(* IEC 61131-3 sources: exOS-Demos/Frameworks/Components/Binary/Sequence/Sequence, 2 files *)

(* ---- Sequence.typ ---- *)
TYPE
	SequenceButtons : 	STRUCT
		ButtonLeft : BOOL;
		ButtonRight : BOOL;
	END_STRUCT;
	Sequence : 	STRUCT
		Buttons : SequenceButtons; (*PUB*)
		Start : BOOL; (*PUB*)
		Active : BOOL; (*SUB*)
	END_STRUCT;
END_TYPE

(* ---- Sequence.fun ---- *)
FUNCTION_BLOCK SequenceInit
	VAR_OUTPUT
		Handle : UDINT;
	END_VAR
	VAR
		_state : USINT;
	END_VAR
END_FUNCTION_BLOCK

FUNCTION_BLOCK SequenceCyclic
	VAR_INPUT
		Enable : BOOL;
		Handle : UDINT;
		Start : BOOL;
		pSequence : REFERENCE TO Sequence;
	END_VAR
	VAR_OUTPUT
		Active : BOOL;
		Error : BOOL;
		Disconnected : BOOL;
		Connected : BOOL;
		Operational : BOOL;
		Aborted : BOOL;
	END_VAR
	VAR
		_state : USINT;
	END_VAR
END_FUNCTION_BLOCK

FUNCTION_BLOCK SequenceExit
	VAR_INPUT
		Handle : UDINT;
	END_VAR
	VAR
		_state : USINT;
	END_VAR
END_FUNCTION_BLOCK
